// Mitsubishi GX Works2 project: 램프2   PLC: Q02/Q02H

PROGRAM MAIN
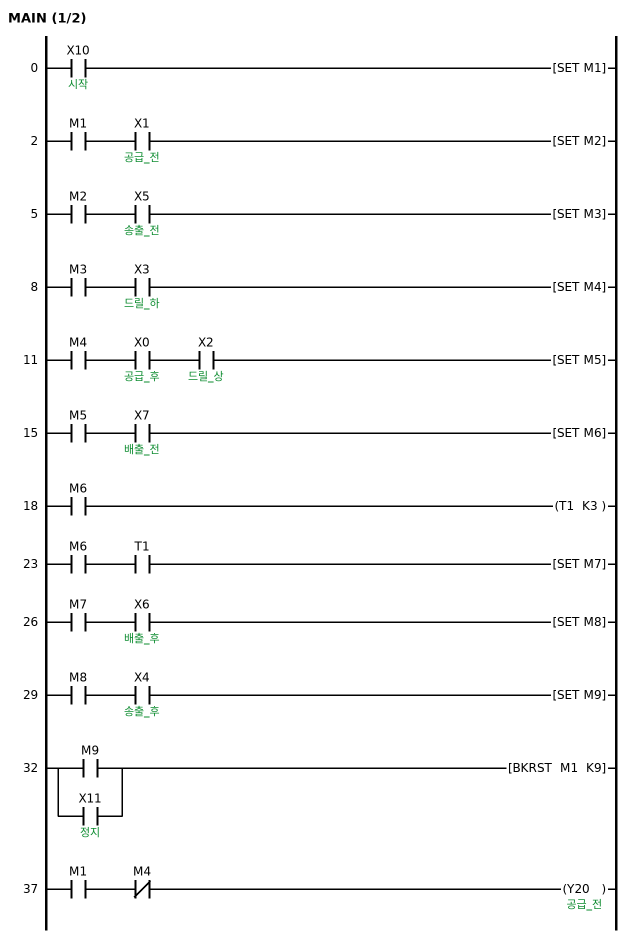
0     LD      X10  ; 시작
      SET     M1
2     LD      M1
      AND     X1  ; 공급_전
      SET     M2
5     LD      M2
      AND     X5  ; 송출_전
      SET     M3
8     LD      M3
      AND     X3  ; 드릴_하
      SET     M4
11    LD      M4
      AND     X0  ; 공급_후
      AND     X2  ; 드릴_상
      SET     M5
15    LD      M5
      AND     X7  ; 배출_전
      SET     M6
18    LD      M6
      OUT     T1 K3
23    LD      M6
      AND     T1
      SET     M7
26    LD      M7
      AND     X6  ; 배출_후
      SET     M8
29    LD      M8
      AND     X4  ; 송출_후
      SET     M9
32    LD      M9
      OR      X11  ; 정지
      BKRST   M1 K9
37    LD      M1
      ANI     M4
      OUT     Y20  ; 공급_전
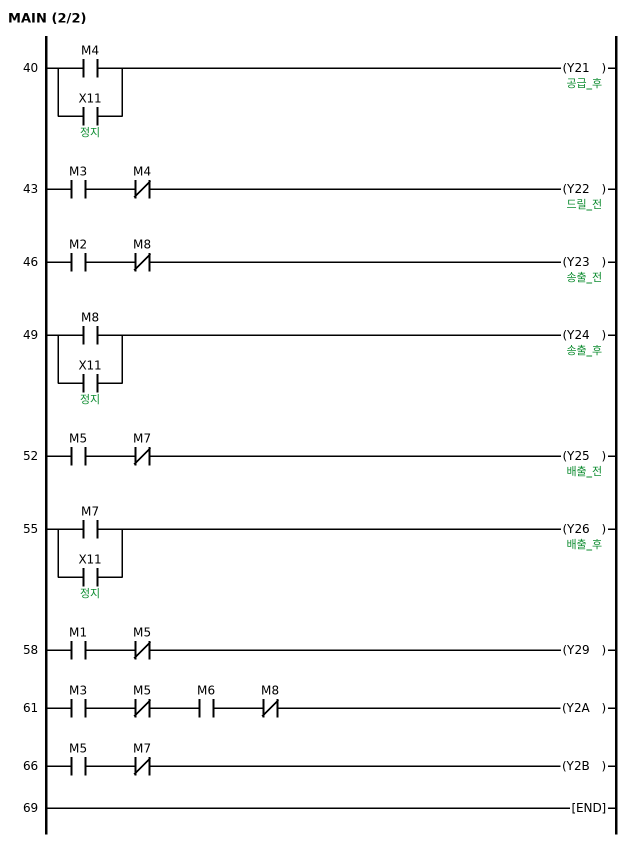
40    LD      M4
      OR      X11  ; 정지
      OUT     Y21  ; 공급_후
43    LD      M3
      ANI     M4
      OUT     Y22  ; 드릴_전
46    LD      M2
      ANI     M8
      OUT     Y23  ; 송출_전
49    LD      M8
      OR      X11  ; 정지
      OUT     Y24  ; 송출_후
52    LD      M5
      ANI     M7
      OUT     Y25  ; 배출_전
55    LD      M7
      OR      X11  ; 정지
      OUT     Y26  ; 배출_후
58    LD      M1
      ANI     M5
      OUT     Y29
61    LD      M3
      ANI     M5
      AND     M6
      ANI     M8
      OUT     Y2A
66    LD      M5
      ANI     M7
      OUT     Y2B
69    END
END_PROGRAM
